# B&R Automation Studio project Autonomous-Robotics-Software-Lab1
Automation Studio 4.5.2.102

## Configuration Config1

### Task classes (Cpu.sw)
```
Cyclic#1:
  Program <- Program.prg
Binaries: udbdef, TCData, ashwd, User, asfw, arconfig, sysconf, Role, ashwac, iomap
Libraries: Library
```

## Logical view

### Library Logical/Library (ANSIC)

#### Library.fun - Exported functions and function blocks
```iecst
{REDUND_ERROR} {REDUND_UNREPLICABLE} FUNCTION_BLOCK FB_integrator (*TODO: Add your comment here*) (*$GROUP=User,$CAT=User,$GROUPICON=User.png,$CATICON=User.png*)
	VAR_INPUT
		in : {REDUND_UNREPLICABLE} REAL;
	END_VAR
	VAR_OUTPUT
		out : {REDUND_UNREPLICABLE} REAL := 0;
	END_VAR
	VAR
		dt : {REDUND_UNREPLICABLE} REAL;
		state : {REDUND_UNREPLICABLE} REAL;
	END_VAR
END_FUNCTION_BLOCK

{REDUND_ERROR} {REDUND_UNREPLICABLE} FUNCTION_BLOCK FB_motor (*TODO: Add your comment here*) (*$GROUP=User,$CAT=User,$GROUPICON=User.png,$CATICON=User.png*)
	VAR_INPUT
		u : {REDUND_UNREPLICABLE} REAL;
	END_VAR
	VAR_OUTPUT
		w : {REDUND_UNREPLICABLE} REAL := 0;
		phi : {REDUND_UNREPLICABLE} REAL;
	END_VAR
	VAR
		integrator : {REDUND_UNREPLICABLE} FB_integrator;
		Tm : {REDUND_UNREPLICABLE} REAL;
		ke : {REDUND_UNREPLICABLE} REAL;
		dt : {REDUND_UNREPLICABLE} REAL;
	END_VAR
END_FUNCTION_BLOCK

{REDUND_ERROR} {REDUND_UNREPLICABLE} FUNCTION_BLOCK FB_Regulator (*TODO: Add your comment here*) (*$GROUP=User,$CAT=User,$GROUPICON=User.png,$CATICON=User.png*)
	VAR_INPUT
		e : {REDUND_UNREPLICABLE} REAL;
	END_VAR
	VAR_OUTPUT
		u : {REDUND_UNREPLICABLE} REAL;
	END_VAR
	VAR
		k_p : {REDUND_UNREPLICABLE} REAL;
		k_i : {REDUND_UNREPLICABLE} REAL;
		integrator : {REDUND_UNREPLICABLE} FB_integrator;
		iyOld : {REDUND_UNREPLICABLE} REAL;
		max_abs_value : {REDUND_UNREPLICABLE} REAL;
		e_p : {REDUND_UNREPLICABLE} REAL;
		dt : {REDUND_UNREPLICABLE} REAL;
	END_VAR
END_FUNCTION_BLOCK
```

#### FB_integrator.c
```c
#include <bur/plctypes.h>
#ifdef __cplusplus
	extern "C"
	{
#endif
#include "Library.h"
#ifdef __cplusplus
	};
#endif
/* TODO: Add your comment here */
void FB_integrator(struct FB_integrator* inst)
{
	inst->out+=inst->in;
}
```

#### FB_motor.c
```c
#include <bur/plctypes.h>
#ifdef __cplusplus
	extern "C"
	{
#endif
#include "Library.h"
#ifdef __cplusplus
	};
#endif
/* TODO: Add your comment here */
void FB_motor(struct FB_motor* inst)
{
	/*TODO: Add your code here*/
	inst->integrator.in = (inst->u*(1/inst->ke) - inst->w)*(inst->dt/inst->Tm);
	FB_integrator(&(inst->integrator));

	inst->w=inst->integrator.out;
	inst->integrator.in=inst->w*inst->dt;
	FB_integrator(&(inst->integrator));

	inst->phi=inst->integrator.out;
}
```

#### FB_Regulator.c
```c
/*
#include <bur/plctypes.h>
#ifdef __cplusplus
	extern "C"
	{
#endif
	#include "Library.h"
#ifdef __cplusplus
	};
#endif
 TODO: Add your comment here
void FB_Regulator(struct FB_Regulator* inst)
{
	//dt = 0.002;
	//k_i = 0.16;
	//k_p = 0.0064;

	REAL a = inst->e * inst->k_p;
	REAL b = inst->e * inst->k_i;
	if (a > 24) a = 24;
	if (a < -24) a = -24;

	inst->integrator.in = b + inst->iyOld;
	FB_integrator(&(inst->integrator));

	REAL sum = a + inst->integrator.out;
	inst->u = sum;
	if (inst->u > inst->max_abs_value) inst->max_abs_value;
	if (inst->u < -inst->max_abs_value) -inst->max_abs_value;
	inst->iyOld = inst->u - sum;

}
*/
#include <bur/plctypes.h>
#ifdef __cplusplus
	extern "C"
	{
#endif
#include "Library.h"
#ifdef __cplusplus
	};
#endif
/* TODO: Add your comment here */
void FB_Regulator(struct FB_Regulator* inst)
{
	/*TODO: Add your code here*/
	inst->integrator.in = inst->e*inst->k_i*inst->dt + inst->iyOld;
	FB_integrator(&(inst->integrator));

	inst->e_p = inst->e*inst->k_p;

	if (inst->e_p < inst->max_abs_value || inst->e_p > -inst->max_abs_value);
	else
	{
		if (inst->e_p > 0) inst->e_p = inst->max_abs_value;
		else inst->e_p = -inst->max_abs_value;
	}

	inst->e_p += inst->integrator.out;
	if (inst->e_p < inst->max_abs_value || inst->e_p > -inst->max_abs_value)
		inst->u = inst->e_p;
	else
	{
		if (inst->e_p > 0) inst->u = inst->max_abs_value;
		else inst ->u = -inst->max_abs_value;
	}

	inst->iyOld = inst->u - inst->e_p;
}
```

### Program Logical/Program (ANSIC)

#### Variables.var
```iecst
VAR
	fb_motor2 : FB_motor;
	fb_controller : FB_Regulator;
	fb_motor : FB_motor;
	speed : REAL;
	Enable : BOOL;
	count : REAL;
	integrator : FB_integrator;
END_VAR
```

#### Cyclic.c
```c
#include <bur/plctypes.h>

#ifdef _DEFAULT_INCLUDES
#include <AsDefault.h>
#endif

void _INIT ProgramInit(void)
{
	Enable=1;
	count=0;
	speed=0;

	fb_motor.dt = 0.01;
	fb_motor.ke=2;
	fb_motor.Tm=0.07;
	fb_motor2.dt=0.01;
	fb_motor2.ke=1;
	fb_motor2.Tm=0.07;

	fb_controller.dt=0.01;
	fb_controller.k_p=1.4;
	fb_controller.k_i=20;
	fb_controller.max_abs_value=24;
}

void _CYCLIC ProgramCyclic(void)
{
	if(Enable == 1)
	{
		count +=10;
		if (count >= 500 && count <= 2000) speed = 40;
		else speed = 5;
	}

	else speed = 0;
	fb_controller.e=speed-fb_motor.w;
	fb_motor2.u=speed*fb_motor2.ke;
	fb_motor.u=fb_controller.u*fb_motor.ke;
	FB_Regulator(&fb_controller);
	FB_motor(&fb_motor);
	FB_motor(&fb_motor2);
}

void _EXIT ProgramExit(void)
{

}
```

Listed in the project but not available here: Logical/Global.typ, Logical/Global.var, Logical/Libraries, Logical/Library/Types.typ, Logical/Library/Constants.var
